PROGRAM P_OutputNonCompensated
VAR
	stValueInput 	: V2Q2u;
	stValueOutput 	: FB_ValveOutput;
END_VAR

stValueInput(
	Ps 	:= G_Sensors.fPressureSupply,
	Pa 	:= G_Simulator.fPistonSidePressure,
	Pb 	:= G_Simulator.fRodSidePressure,
	y 	:= G_Work.fJoystickY,
	u	=> stValueOutput.fNormalizedInput
);

END_PROGRAM

(* stored: Version 1.1.0.1, ProductVersion 3.1.4024.13
   POU P_OutputNonCompensated: Id {91e8730f-330f-4841-8441-0d9eae6d44e6}, SpecialFunc None *)
